{attribute 'GeneratedUsingTerminal: EK1122-0000-0018'}
{attribute addProperty BoxType "EK1122-0000-0018"}
{attribute addProperty Id "Beckhoff_EL7xxxsub_EK1100EK1100_1FC0878B2"}
{attribute addProperty CRC "4284980018"}
{attribute addProperty Size "2"}
TYPE Beckhoff_EL7xxxEK1122_FF679B32 EXTENDS EK1122_1FC0878B :
STRUCT
	{attribute addProperty Name "Beckhoff_EL7xxxsub_EK1100"}
	{attribute addProperty PreviousPort "Beckhoff EL7xxxEK1122 : D"}
	Beckhoff_EL7xxxsub_EK1100 : EK1100_1FC0878B;
END_STRUCT
END_TYPE

(* stored: Version 1.2.0.0, ProductVersion 3.1.4024.9
   DUT Beckhoff_EL7xxxEK1122_FF679B32: Id {53411c86-2f61-4272-a145-c1a2c8bbbd2b} *)
